// LS Electric XG5000 project: 220021116_CEP_XG500
// PLC NewPLC

PROGRAM NewProgram (task: Scan Program)

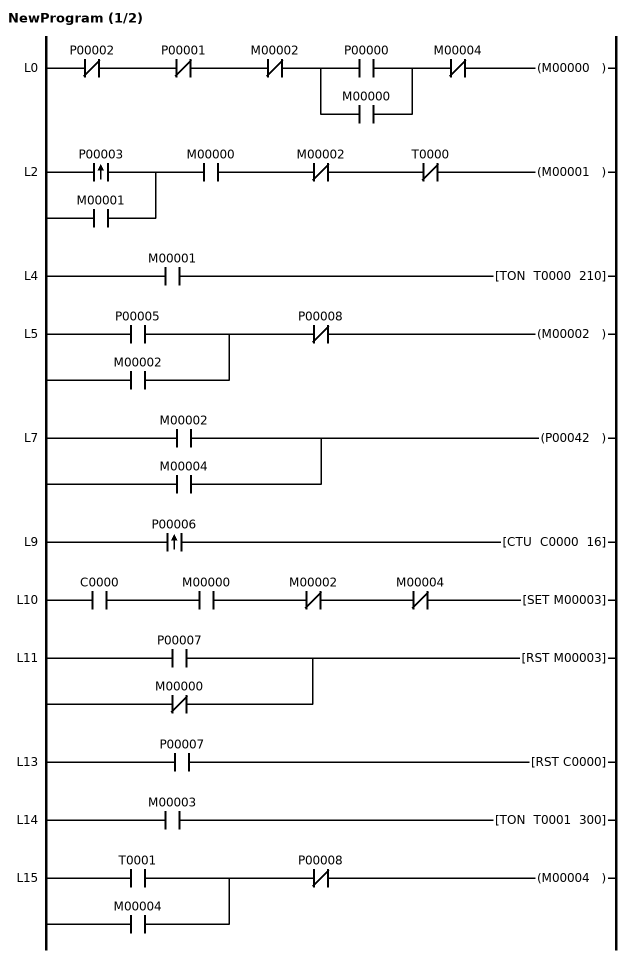
; L0
LOAD NOT  P00002
AND NOT   P00001
AND NOT   M00002
LOAD      P00000
OR        M00000
AND LOAD
AND NOT   M00004
OUT       M00000
; L2
LOADP     P00003
OR        M00001
AND       M00000
AND NOT   M00002
AND NOT   T0000
OUT       M00001
; L4
LOAD      M00001
TON       T0000 210
; L5
LOAD      P00005
OR        M00002
AND NOT   P00008
OUT       M00002
; L7
LOAD      M00002
OR        M00004
OUT       P00042
; L9
LOADP     P00006
CTU       C0000 16
; L10
LOAD      C0000
AND       M00000
AND NOT   M00002
AND NOT   M00004
SET       M00003
; L11
LOAD      P00007
OR NOT    M00000
RST       M00003
; L13
LOAD      P00007
RST       C0000
; L14
LOAD      M00003
TON       T0001 300
; L15
LOAD      T0001
OR        M00004
AND NOT   P00008
OUT       M00004

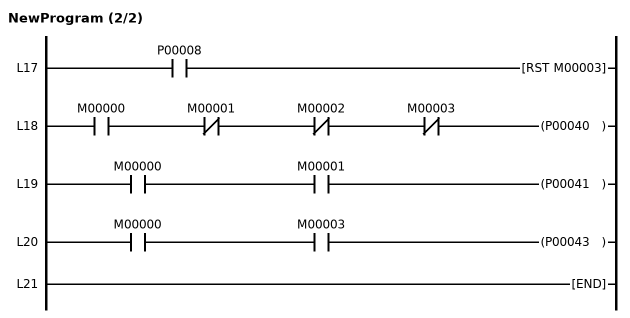
; L17
LOAD      P00008
RST       M00003
; L18
LOAD      M00000
AND NOT   M00001
AND NOT   M00002
AND NOT   M00003
OUT       P00040
; L19
LOAD      M00000
AND       M00001
OUT       P00041
; L20
LOAD      M00000
AND       M00003
OUT       P00043
; L21
END